// TIA Portal V16 export
// export: Created 2022-11-14T17:35:29.4919195Z, ExportSetting WithDefaults, DisplayName Totally Integrated Automation Portal, DisplayVersion V16, DisplayName TIA Portal Version Control Interface, DisplayVersion V16, DisplayName TIA Portal Openness, DisplayVersion V16, DisplayName STEP 7 Professional, DisplayVersion V16, DisplayName STEP 7 Safety, DisplayVersion V16, DisplayName WinCC Advanced, DisplayVersion V16
FUNCTION "FC41_NoRopeUnit" : Void   // FC41, LAD
TITLE = No rope unit
{ S7_Optimized_Access := 'FALSE' }
AUTHOR : Robopac
VERSION : 0.0
// stored: AutoNumber false, IsIECCheckEnabled false, SetENOAutomatically false, UDAEnableTagReadback false
BEGIN

REGION Network 1: RopeUnitOk1: Rope unit open
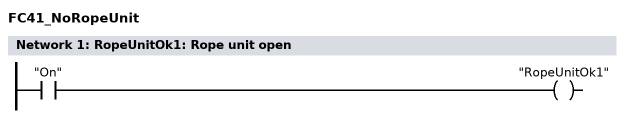
   RUNG wire#powerrail
      Contact( "On" )
      Coil( "RopeUnitOk1" )
   END_RUNG
   // the same network as SCL:
   "RopeUnitOk1" := "On";
END_REGION
END_FUNCTION
